Staubli VAL3: newProject1.dtx

public frame fUserFrame = {x=480, y=190, z=-101.4, rx=2, rz=-90, fatherId=world[0]}
public jointRx jtPark = {j1=-90, j2=-20, j3=130, j5=-60, j6=178}
public mdesc mNomSpeed = {blend=off}
public mdesc mdJointBlend = {accel=250, decel=150, leave=1, reach=1}
public mdesc mdLineBlend = {accel=80, vel=50, decel=50, tmax=100, rmax=9999, leave=2, reach=2}
public pointRx ptRoutingPath[478]
  [0] = {x=50.46, y=-3.411, z=224.779, rx=180, ry=-42.407, rz=-159.872, shoulder=lefty, elbow=epositive, wrist=wpositive, fatherId=fUserFrame[0]}
  [1] = {x=4.278, y=-3.411, z=174.216, rx=180, ry=-42.407, rz=-159.872, shoulder=lefty, elbow=epositive, wrist=wpositive, fatherId=fUserFrame[0]}
  [2] = {x=4.278, y=-3.411, z=124.216, rx=180, ry=-42.407, rz=-159.872, shoulder=lefty, elbow=epositive, wrist=wpositive, fatherId=fUserFrame[0]}
  [3] = {x=3.791, y=1.027, z=124.278, rx=180, ry=-42.212, rz=-156.401, shoulder=lefty, elbow=epositive, wrist=wpositive, fatherId=fUserFrame[0]}
  [4] = {x=4.289, y=5.504, z=124.132, rx=180, ry=-42.386, rz=-152.9, shoulder=lefty, elbow=epositive, wrist=wpositive, fatherId=fUserFrame[0]}
  [5] = {x=5.782, y=9.947, z=123.764, rx=180, ry=-42.934, rz=-149.41, shoulder=lefty, elbow=epositive, wrist=wpositive, fatherId=fUserFrame[0]}
  [6] = {x=8.224, y=14.41, z=123.139, rx=180, ry=-43.84, rz=-145.883, shoulder=lefty, elbow=epositive, wrist=wpositive, fatherId=fUserFrame[0]}
  [7] = {x=11.501, y=18.894, z=122.2, rx=180, ry=-45.057, rz=-142.303, shoulder=lefty, elbow=epositive, wrist=wpositive, fatherId=fUserFrame[0]}
  [8] = {x=9.824, y=14.861, z=122.959, rx=180, ry=-44.571, rz=-145.522, shoulder=lefty, elbow=epositive, wrist=wpositive, fatherId=fUserFrame[0]}
  [9] = {x=8.613, y=10.87, z=123.51, rx=180, ry=-44.23, rz=-148.678, shoulder=lefty, elbow=epositive, wrist=wpositive, fatherId=fUserFrame[0]}
  [10] = {x=7.921, y=6.919, z=123.87, rx=180, ry=-44.06, rz=-151.783, shoulder=lefty, elbow=epositive, wrist=wpositive, fatherId=fUserFrame[0]}
  [11] = {x=7.772, y=2.954, z=124.054, rx=180, ry=-44.073, rz=-154.884, shoulder=lefty, elbow=epositive, wrist=wpositive, fatherId=fUserFrame[0]}
  [12] = {x=8.16, y=-0.997, z=124.064, rx=180, ry=-44.266, rz=-157.97, shoulder=lefty, elbow=epositive, wrist=wpositive, fatherId=fUserFrame[0]}
  [13] = {x=7.987, y=2.551, z=124.05, rx=180, ry=-44.179, rz=-155.198, shoulder=lefty, elbow=epositive, wrist=wpositive, fatherId=fUserFrame[0]}
  [14] = {x=8.556, y=6.099, z=123.875, rx=180, ry=-44.383, rz=-152.423, shoulder=lefty, elbow=epositive, wrist=wpositive, fatherId=fUserFrame[0]}
  [15] = {x=9.86, y=9.613, z=123.529, rx=180, ry=-44.879, rz=-149.664, shoulder=lefty, elbow=epositive, wrist=wpositive, fatherId=fUserFrame[0]}
  [16] = {x=11.866, y=13.123, z=122.992, rx=180, ry=-45.653, rz=-146.893, shoulder=lefty, elbow=epositive, wrist=wpositive, fatherId=fUserFrame[0]}
  [17] = {x=14.502, y=16.628, z=122.234, rx=180, ry=-46.679, rz=-144.107, shoulder=lefty, elbow=epositive, wrist=wpositive, fatherId=fUserFrame[0]}
  [18] = {x=17.496, y=20.822, z=121.12, rx=180, ry=-47.769, rz=-140.737, shoulder=lefty, elbow=epositive, wrist=wpositive, fatherId=fUserFrame[0]}
  [19] = {x=20.739, y=24.824, z=119.755, rx=180, ry=-48.936, rz=-137.46, shoulder=lefty, elbow=epositive, wrist=wpositive, fatherId=fUserFrame[0]}
  [20] = {x=24.162, y=28.607, z=118.15, rx=180, ry=-50.165, rz=-134.293, shoulder=lefty, elbow=epositive, wrist=wpositive, fatherId=fUserFrame[0]}
  [21] = {x=27.716, y=32.196, z=116.305, rx=180, ry=-51.442, rz=-131.213, shoulder=lefty, elbow=epositive, wrist=wpositive, fatherId=fUserFrame[0]}
  [22] = {x=31.353, y=35.61, z=114.221, rx=180, ry=-52.756, rz=-128.203, shoulder=lefty, elbow=epositive, wrist=wpositive, fatherId=fUserFrame[0]}
  [23] = {x=35.033, y=38.861, z=111.903, rx=180, ry=-54.096, rz=-125.249, shoulder=lefty, elbow=epositive, wrist=wpositive, fatherId=fUserFrame[0]}
  [24] = {x=38.719, y=41.93, z=109.366, rx=180, ry=-55.456, rz=-122.365, shoulder=lefty, elbow=epositive, wrist=wpositive, fatherId=fUserFrame[0]}
  [25] = {x=42.278, y=44.785, z=106.677, rx=180, ry=-56.784, rz=-119.579, shoulder=lefty, elbow=epositive, wrist=wpositive, fatherId=fUserFrame[0]}
  [26] = {x=45.697, y=47.475, z=103.838, rx=180, ry=-58.069, rz=-116.85, shoulder=lefty, elbow=epositive, wrist=wpositive, fatherId=fUserFrame[0]}
  [27] = {x=49.013, y=50.027, z=100.834, rx=180, ry=-59.331, rz=-114.154, shoulder=lefty, elbow=epositive, wrist=wpositive, fatherId=fUserFrame[0]}
  [28] = {x=44.083, y=48.91, z=103.812, rx=180, ry=-56.777, rz=-115.386, shoulder=lefty, elbow=epositive, wrist=wpositive, fatherId=fUserFrame[0]}
  [29] = {x=38.578, y=47.741, z=106.69, rx=180, ry=-54.005, rz=-116.65, shoulder=lefty, elbow=epositive, wrist=wpositive, fatherId=fUserFrame[0]}
  [30] = {x=33.15, y=46.43, z=109.226, rx=180, ry=-51.395, rz=-118.029, shoulder=lefty, elbow=epositive, wrist=wpositive, fatherId=fUserFrame[0]}
  [31] = {x=27.673, y=45.016, z=111.467, rx=180, ry=-48.846, rz=-119.479, shoulder=lefty, elbow=epositive, wrist=wpositive, fatherId=fUserFrame[0]}
  [32] = {x=22.349, y=43.394, z=113.421, rx=180, ry=-46.48, rz=-121.092, shoulder=lefty, elbow=epositive, wrist=wpositive, fatherId=fUserFrame[0]}
  [33] = {x=16.731, y=41.59, z=115.171, rx=180, ry=-44.042, rz=-122.836, shoulder=lefty, elbow=epositive, wrist=wpositive, fatherId=fUserFrame[0]}
  [34] = {x=10.985, y=39.551, z=116.679, rx=180, ry=-41.623, rz=-124.751, shoulder=lefty, elbow=epositive, wrist=wpositive, fatherId=fUserFrame[0]}
  [35] = {x=5.01, y=37.376, z=117.894, rx=180, ry=-39.136, rz=-126.747, shoulder=lefty, elbow=epositive, wrist=wpositive, fatherId=fUserFrame[0]}
  [36] = {x=-0.804, y=35.019, z=118.802, rx=180, ry=-36.769, rz=-128.86, shoulder=lefty, elbow=epositive, wrist=wpositive, fatherId=fUserFrame[0]}
  [37] = {x=-6.341, y=32.513, z=119.42, rx=180, ry=-34.555, rz=-131.058, shoulder=lefty, elbow=epositive, wrist=wpositive, fatherId=fUserFrame[0]}
  [38] = {x=-11.541, y=29.826, z=119.795, rx=180, ry=-32.512, rz=-133.367, shoulder=lefty, elbow=epositive, wrist=wpositive, fatherId=fUserFrame[0]}
  [39] = {x=-16.328, y=26.961, z=119.972, rx=180, ry=-30.663, rz=-135.78, shoulder=lefty, elbow=epositive, wrist=wpositive, fatherId=fUserFrame[0]}
  [40] = {x=-20.759, y=23.89, z=119.984, rx=180, ry=-28.97, rz=-138.319, shoulder=lefty, elbow=epositive, wrist=wpositive, fatherId=fUserFrame[0]}
  [41] = {x=-24.662, y=20.615, z=119.891, rx=180, ry=-27.501, rz=-140.98, shoulder=lefty, elbow=epositive, wrist=wpositive, fatherId=fUserFrame[0]}
  [42] = {x=-28.137, y=17.281, z=119.682, rx=180, ry=-26.181, rz=-143.656, shoulder=lefty, elbow=epositive, wrist=wpositive, fatherId=fUserFrame[0]}
  [43] = {x=-30.954, y=14.026, z=119.435, rx=180, ry=-25.107, rz=-146.251, shoulder=lefty, elbow=epositive, wrist=wpositive, fatherId=fUserFrame[0]}
  [44] = {x=-33.378, y=10.884, z=119.125, rx=180, ry=-24.152, rz=-148.747, shoulder=lefty, elbow=epositive, wrist=wpositive, fatherId=fUserFrame[0]}
  [45] = {x=-35.18, y=7.837, z=118.856, rx=180, ry=-23.436, rz=-151.164, shoulder=lefty, elbow=epositive, wrist=wpositive, fatherId=fUserFrame[0]}
  [46] = {x=-36.701, y=4.771, z=118.561, rx=180, ry=-22.799, rz=-153.585, shoulder=lefty, elbow=epositive, wrist=wpositive, fatherId=fUserFrame[0]}
  [47] = {x=-37.634, y=1.68, z=118.351, rx=180, ry=-22.393, rz=-156.021, shoulder=lefty, elbow=epositive, wrist=wpositive, fatherId=fUserFrame[0]}
  [48] = {x=-31.685, y=1.329, z=120.133, rx=180, ry=-25.334, rz=-156.276, shoulder=lefty, elbow=epositive, wrist=wpositive, fatherId=fUserFrame[0]}
  [49] = {x=-28.486, y=1.091, z=120.955, rx=180, ry=-26.896, rz=-156.452, shoulder=lefty, elbow=epositive, wrist=wpositive, fatherId=fUserFrame[0]}
  [50] = {x=-25.13, y=0.851, z=121.716, rx=180, ry=-28.521, rz=-156.629, shoulder=lefty, elbow=epositive, wrist=wpositive, fatherId=fUserFrame[0]}
  [51] = {x=-21.648, y=0.56, z=122.401, rx=180, ry=-30.194, rz=-156.845, shoulder=lefty, elbow=epositive, wrist=wpositive, fatherId=fUserFrame[0]}
  [52] = {x=-17.999, y=0.268, z=123.005, rx=180, ry=-31.937, rz=-157.062, shoulder=lefty, elbow=epositive, wrist=wpositive, fatherId=fUserFrame[0]}
  [53] = {x=-14.2, y=-0.07, z=123.512, rx=180, ry=-33.74, rz=-157.314, shoulder=lefty, elbow=epositive, wrist=wpositive, fatherId=fUserFrame[0]}
  [54] = {x=-10.214, y=-0.41, z=123.912, rx=180, ry=-35.624, rz=-157.568, shoulder=lefty, elbow=epositive, wrist=wpositive, fatherId=fUserFrame[0]}
  [55] = {x=-6.064, y=-0.79, z=124.188, rx=180, ry=-37.576, rz=-157.852, shoulder=lefty, elbow=epositive, wrist=wpositive, fatherId=fUserFrame[0]}
  [56] = {x=-1.901, y=-1.162, z=124.321, rx=180, ry=-39.531, rz=-158.13, shoulder=lefty, elbow=epositive, wrist=wpositive, fatherId=fUserFrame[0]}
  [57] = {x=2.184, y=-1.553, z=124.312, rx=180, ry=-41.448, rz=-158.423, shoulder=lefty, elbow=epositive, wrist=wpositive, fatherId=fUserFrame[0]}
  [58] = {x=6.214, y=-1.935, z=124.167, rx=180, ry=-43.341, rz=-158.71, shoulder=lefty, elbow=epositive, wrist=wpositive, fatherId=fUserFrame[0]}
  [59] = {x=10.181, y=-2.334, z=123.892, rx=180, ry=-45.206, rz=-159.01, shoulder=lefty, elbow=epositive, wrist=wpositive, fatherId=fUserFrame[0]}
  [60] = {x=14.101, y=-2.726, z=123.491, rx=180, ry=-47.055, rz=-159.305, shoulder=lefty, elbow=epositive, wrist=wpositive, fatherId=fUserFrame[0]}
  [61] = {x=17.978, y=-3.133, z=122.966, rx=180, ry=-48.89, rz=-159.612, shoulder=lefty, elbow=epositive, wrist=wpositive, fatherId=fUserFrame[0]}
  [62] = {x=21.827, y=-3.535, z=122.317, rx=180, ry=-50.72, rz=-159.914, shoulder=lefty, elbow=epositive, wrist=wpositive, fatherId=fUserFrame[0]}
  [63] = {x=25.648, y=-3.944, z=121.544, rx=180, ry=-52.547, rz=-160.223, shoulder=lefty, elbow=epositive, wrist=wpositive, fatherId=fUserFrame[0]}
  [64] = {x=29.434, y=-4.346, z=120.65, rx=180, ry=-54.37, rz=-160.526, shoulder=lefty, elbow=epositive, wrist=wpositive, fatherId=fUserFrame[0]}
  [65] = {x=33.191, y=-4.75, z=119.634, rx=180, ry=-56.193, rz=-160.831, shoulder=lefty, elbow=epositive, wrist=wpositive, fatherId=fUserFrame[0]}
  [66] = {x=36.907, y=-5.147, z=118.499, rx=180, ry=-58.013, rz=-161.131, shoulder=lefty, elbow=epositive, wrist=wpositive, fatherId=fUserFrame[0]}
  [67] = {x=36.9, y=-1.421, z=118.608, rx=180, ry=-58.063, rz=-158.213, shoulder=lefty, elbow=epositive, wrist=wpositive, fatherId=fUserFrame[0]}
  [68] = {x=36.824, y=2.407, z=118.608, rx=180, ry=-58.029, rz=-155.227, shoulder=lefty, elbow=epositive, wrist=wpositive, fatherId=fUserFrame[0]}
  [69] = {x=36.718, y=6.276, z=118.48, rx=180, ry=-57.927, rz=-152.208, shoulder=lefty, elbow=epositive, wrist=wpositive, fatherId=fUserFrame[0]}
  [70] = {x=36.616, y=10.149, z=118.211, rx=180, ry=-57.771, rz=-149.173, shoulder=lefty, elbow=epositive, wrist=wpositive, fatherId=fUserFrame[0]}
  [71] = {x=36.51, y=14.016, z=117.804, rx=180, ry=-57.557, rz=-146.122, shoulder=lefty, elbow=epositive, wrist=wpositive, fatherId=fUserFrame[0]}
  [72] = {x=37.169, y=16.535, z=117.228, rx=180, ry=-57.751, rz=-144.116, shoulder=lefty, elbow=epositive, wrist=wpositive, fatherId=fUserFrame[0]}
  [73] = {x=38.02, y=19.029, z=116.525, rx=180, ry=-58.02, rz=-142.115, shoulder=lefty, elbow=epositive, wrist=wpositive, fatherId=fUserFrame[0]}
  [74] = {x=38.787, y=21.476, z=115.79, rx=180, ry=-58.228, rz=-140.133, shoulder=lefty, elbow=epositive, wrist=wpositive, fatherId=fUserFrame[0]}
  [75] = {x=39.708, y=23.854, z=114.947, rx=180, ry=-58.501, rz=-138.184, shoulder=lefty, elbow=epositive, wrist=wpositive, fatherId=fUserFrame[0]}
  [76] = {x=40.535, y=26.179, z=114.082, rx=180, ry=-58.709, rz=-136.254, shoulder=lefty, elbow=epositive, wrist=wpositive, fatherId=fUserFrame[0]}
  [77] = {x=41.497, y=28.44, z=113.115, rx=180, ry=-58.976, rz=-134.351, shoulder=lefty, elbow=epositive, wrist=wpositive, fatherId=fUserFrame[0]}
  [78] = {x=42.362, y=30.659, z=112.13, rx=180, ry=-59.176, rz=-132.457, shoulder=lefty, elbow=epositive, wrist=wpositive, fatherId=fUserFrame[0]}
  [79] = {x=43.343, y=32.818, z=111.05, rx=180, ry=-59.428, rz=-130.584, shoulder=lefty, elbow=epositive, wrist=wpositive, fatherId=fUserFrame[0]}
  [80] = {x=44.221, y=34.939, z=109.958, rx=180, ry=-59.61, rz=-128.715, shoulder=lefty, elbow=epositive, wrist=wpositive, fatherId=fUserFrame[0]}
  [81] = {x=45.196, y=37.004, z=108.778, rx=180, ry=-59.834, rz=-126.861, shoulder=lefty, elbow=epositive, wrist=wpositive, fatherId=fUserFrame[0]}
  [82] = {x=46.064, y=39.037, z=107.59, rx=180, ry=-59.985, rz=-125.002, shoulder=lefty, elbow=epositive, wrist=wpositive, fatherId=fUserFrame[0]}
  [83] = {x=47.013, y=41.002, z=106.326, rx=180, ry=-60.173, rz=-123.166, shoulder=lefty, elbow=epositive, wrist=wpositive, fatherId=fUserFrame[0]}
  [84] = {x=47.863, y=42.921, z=105.062, rx=180, ry=-60.293, rz=-121.334, shoulder=lefty, elbow=epositive, wrist=wpositive, fatherId=fUserFrame[0]}
  [85] = {x=48.809, y=44.772, z=103.716, rx=180, ry=-60.46, rz=-119.524, shoulder=lefty, elbow=epositive, wrist=wpositive, fatherId=fUserFrame[0]}
  [86] = {x=49.686, y=46.591, z=102.355, rx=180, ry=-60.572, rz=-117.702, shoulder=lefty, elbow=epositive, wrist=wpositive, fatherId=fUserFrame[0]}
  [87] = {x=50.7, y=48.352, z=100.888, rx=180, ry=-60.754, rz=-115.891, shoulder=lefty, elbow=epositive, wrist=wpositive, fatherId=fUserFrame[0]}
  [88] = {x=51.727, y=50.068, z=99.369, rx=180, ry=-60.931, rz=-114.077, shoulder=lefty, elbow=epositive, wrist=wpositive, fatherId=fUserFrame[0]}
  [89] = {x=52.948, y=51.706, z=97.716, rx=180, ry=-61.221, rz=-112.29, shoulder=lefty, elbow=epositive, wrist=wpositive, fatherId=fUserFrame[0]}
  [90] = {x=54.179, y=53.292, z=96.009, rx=180, ry=-61.51, rz=-110.505, shoulder=lefty, elbow=epositive, wrist=wpositive, fatherId=fUserFrame[0]}
  [91] = {x=55.616, y=54.796, z=94.148, rx=180, ry=-61.931, rz=-108.75, shoulder=lefty, elbow=epositive, wrist=wpositive, fatherId=fUserFrame[0]}
  [92] = {x=52.563, y=54.509, z=96.159, rx=180, ry=-60.128, rz=-109.12, shoulder=lefty, elbow=epositive, wrist=wpositive, fatherId=fUserFrame[0]}
  [93] = {x=47.423, y=53.901, z=99.331, rx=180, ry=-57.206, rz=-109.889, shoulder=lefty, elbow=epositive, wrist=wpositive, fatherId=fUserFrame[0]}
  [94] = {x=44.683, y=53.582, z=100.858, rx=180, ry=-55.691, rz=-110.285, shoulder=lefty, elbow=epositive, wrist=wpositive, fatherId=fUserFrame[0]}
  [95] = {x=41.917, y=53.209, z=102.324, rx=180, ry=-54.209, rz=-110.738, shoulder=lefty, elbow=epositive, wrist=wpositive, fatherId=fUserFrame[0]}
  [96] = {x=38.974, y=52.828, z=103.762, rx=180, ry=-52.655, rz=-111.197, shoulder=lefty, elbow=epositive, wrist=wpositive, fatherId=fUserFrame[0]}
  [97] = {x=36.005, y=52.436, z=105.108, rx=180, ry=-51.115, rz=-111.665, shoulder=lefty, elbow=epositive, wrist=wpositive, fatherId=fUserFrame[0]}
  [98] = {x=33.04, y=52.03, z=106.355, rx=180, ry=-49.603, rz=-112.143, shoulder=lefty, elbow=epositive, wrist=wpositive, fatherId=fUserFrame[0]}
  [99] = {x=27.328, y=51.09, z=108.557, rx=180, ry=-46.799, rz=-113.223, shoulder=lefty, elbow=epositive, wrist=wpositive, fatherId=fUserFrame[0]}
  [100] = {x=21.384, y=50.082, z=110.477, rx=180, ry=-43.956, rz=-114.355, shoulder=lefty, elbow=epositive, wrist=wpositive, fatherId=fUserFrame[0]}
  [101] = {x=18.339, y=49.516, z=111.339, rx=180, ry=-42.539, rz=-114.977, shoulder=lefty, elbow=epositive, wrist=wpositive, fatherId=fUserFrame[0]}
  [102] = {x=15.169, y=48.922, z=112.135, rx=180, ry=-41.078, rz=-115.621, shoulder=lefty, elbow=epositive, wrist=wpositive, fatherId=fUserFrame[0]}
  [103] = {x=11.868, y=48.297, z=112.858, rx=180, ry=-39.57, rz=-116.289, shoulder=lefty, elbow=epositive, wrist=wpositive, fatherId=fUserFrame[0]}
  [104] = {x=8.507, y=47.631, z=113.495, rx=180, ry=-38.055, rz=-116.989, shoulder=lefty, elbow=epositive, wrist=wpositive, fatherId=fUserFrame[0]}
  [105] = {x=5.171, y=46.89, z=114.053, rx=180, ry=-36.584, rz=-117.755, shoulder=lefty, elbow=epositive, wrist=wpositive, fatherId=fUserFrame[0]}
  [106] = {x=1.817, y=46.093, z=114.527, rx=180, ry=-35.126, rz=-118.565, shoulder=lefty, elbow=epositive, wrist=wpositive, fatherId=fUserFrame[0]}
  [107] = {x=-1.542, y=45.234, z=114.917, rx=180, ry=-33.688, rz=-119.423, shoulder=lefty, elbow=epositive, wrist=wpositive, fatherId=fUserFrame[0]}
  [108] = {x=-4.897, y=44.308, z=115.225, rx=180, ry=-32.273, rz=-120.333, shoulder=lefty, elbow=epositive, wrist=wpositive, fatherId=fUserFrame[0]}
  [109] = {x=-11.566, y=42.2, z=115.614, rx=180, ry=-29.532, rz=-122.352, shoulder=lefty, elbow=epositive, wrist=wpositive, fatherId=fUserFrame[0]}
  [110] = {x=-17.965, y=39.906, z=115.675, rx=180, ry=-26.955, rz=-124.491, shoulder=lefty, elbow=epositive, wrist=wpositive, fatherId=fUserFrame[0]}
  [111] = {x=-24.031, y=37.42, z=115.459, rx=180, ry=-24.556, rz=-126.753, shoulder=lefty, elbow=epositive, wrist=wpositive, fatherId=fUserFrame[0]}
  [112] = {x=-29.593, y=34.771, z=115.041, rx=180, ry=-22.399, rz=-129.107, shoulder=lefty, elbow=epositive, wrist=wpositive, fatherId=fUserFrame[0]}
  [113] = {x=-34.725, y=31.939, z=114.463, rx=180, ry=-20.436, rz=-131.569, shoulder=lefty, elbow=epositive, wrist=wpositive, fatherId=fUserFrame[0]}
  [114] = {x=-39.297, y=28.891, z=113.822, rx=180, ry=-18.731, rz=-134.16, shoulder=lefty, elbow=epositive, wrist=wpositive, fatherId=fUserFrame[0]}
  [115] = {x=-43.448, y=25.6, z=113.12, rx=180, ry=-17.202, rz=-136.9, shoulder=lefty, elbow=epositive, wrist=wpositive, fatherId=fUserFrame[0]}
  [116] = {x=-47.036, y=22.037, z=112.449, rx=180, ry=-15.915, rz=-139.808, shoulder=lefty, elbow=epositive, wrist=wpositive, fatherId=fUserFrame[0]}
  [117] = {x=-50.183, y=18.336, z=111.758, rx=180, ry=-14.774, rz=-142.782, shoulder=lefty, elbow=epositive, wrist=wpositive, fatherId=fUserFrame[0]}
  [118] = {x=-52.715, y=14.806, z=111.116, rx=180, ry=-13.835, rz=-145.601, shoulder=lefty, elbow=epositive, wrist=wpositive, fatherId=fUserFrame[0]}
  [119] = {x=-52.715, y=14.806, z=161.116, rx=180, ry=-13.835, rz=-145.601, shoulder=lefty, elbow=epositive, wrist=wpositive, fatherId=fUserFrame[0]}
  [120] = {x=4.278, y=3.411, z=174.216, rx=180, ry=-42.407, rz=159.872, shoulder=lefty, elbow=epositive, wrist=wpositive, fatherId=fUserFrame[0]}
  [121] = {x=4.278, y=3.411, z=124.216, rx=180, ry=-42.407, rz=159.872, shoulder=lefty, elbow=epositive, wrist=wpositive, fatherId=fUserFrame[0]}
  [122] = {x=3.791, y=-1.027, z=124.278, rx=180, ry=-42.212, rz=156.401, shoulder=lefty, elbow=epositive, wrist=wpositive, fatherId=fUserFrame[0]}
  [123] = {x=4.289, y=-5.504, z=124.132, rx=180, ry=-42.386, rz=152.9, shoulder=lefty, elbow=epositive, wrist=wpositive, fatherId=fUserFrame[0]}
  [124] = {x=5.782, y=-9.947, z=123.764, rx=180, ry=-42.934, rz=149.41, shoulder=lefty, elbow=epositive, wrist=wpositive, fatherId=fUserFrame[0]}
  [125] = {x=8.224, y=-14.41, z=123.139, rx=180, ry=-43.84, rz=145.883, shoulder=lefty, elbow=epositive, wrist=wpositive, fatherId=fUserFrame[0]}
  [126] = {x=11.501, y=-18.894, z=122.2, rx=180, ry=-45.057, rz=142.303, shoulder=lefty, elbow=epositive, wrist=wpositive, fatherId=fUserFrame[0]}
  [127] = {x=9.824, y=-14.861, z=122.959, rx=180, ry=-44.571, rz=145.522, shoulder=lefty, elbow=epositive, wrist=wpositive, fatherId=fUserFrame[0]}
  [128] = {x=8.613, y=-10.87, z=123.51, rx=180, ry=-44.23, rz=148.678, shoulder=lefty, elbow=epositive, wrist=wpositive, fatherId=fUserFrame[0]}
  [129] = {x=7.921, y=-6.919, z=123.87, rx=180, ry=-44.06, rz=151.783, shoulder=lefty, elbow=epositive, wrist=wpositive, fatherId=fUserFrame[0]}
  [130] = {x=7.772, y=-2.954, z=124.054, rx=180, ry=-44.073, rz=154.884, shoulder=lefty, elbow=epositive, wrist=wpositive, fatherId=fUserFrame[0]}
  [131] = {x=8.16, y=0.997, z=124.064, rx=180, ry=-44.266, rz=157.97, shoulder=lefty, elbow=epositive, wrist=wpositive, fatherId=fUserFrame[0]}
  [132] = {x=7.987, y=-2.551, z=124.05, rx=180, ry=-44.179, rz=155.198, shoulder=lefty, elbow=epositive, wrist=wpositive, fatherId=fUserFrame[0]}
  [133] = {x=8.556, y=-6.099, z=123.875, rx=180, ry=-44.383, rz=152.423, shoulder=lefty, elbow=epositive, wrist=wpositive, fatherId=fUserFrame[0]}
  [134] = {x=9.86, y=-9.613, z=123.529, rx=180, ry=-44.879, rz=149.664, shoulder=lefty, elbow=epositive, wrist=wpositive, fatherId=fUserFrame[0]}
  [135] = {x=11.866, y=-13.123, z=122.992, rx=180, ry=-45.653, rz=146.893, shoulder=lefty, elbow=epositive, wrist=wpositive, fatherId=fUserFrame[0]}
  [136] = {x=14.502, y=-16.628, z=122.234, rx=180, ry=-46.679, rz=144.107, shoulder=lefty, elbow=epositive, wrist=wpositive, fatherId=fUserFrame[0]}
  [137] = {x=17.496, y=-20.822, z=121.12, rx=180, ry=-47.769, rz=140.737, shoulder=lefty, elbow=epositive, wrist=wpositive, fatherId=fUserFrame[0]}
  [138] = {x=20.739, y=-24.824, z=119.755, rx=180, ry=-48.936, rz=137.46, shoulder=lefty, elbow=epositive, wrist=wpositive, fatherId=fUserFrame[0]}
  [139] = {x=24.162, y=-28.607, z=118.15, rx=180, ry=-50.165, rz=134.293, shoulder=lefty, elbow=epositive, wrist=wpositive, fatherId=fUserFrame[0]}
  [140] = {x=27.716, y=-32.196, z=116.305, rx=180, ry=-51.442, rz=131.213, shoulder=lefty, elbow=epositive, wrist=wpositive, fatherId=fUserFrame[0]}
  [141] = {x=31.353, y=-35.61, z=114.221, rx=180, ry=-52.756, rz=128.203, shoulder=lefty, elbow=epositive, wrist=wpositive, fatherId=fUserFrame[0]}
  [142] = {x=35.033, y=-38.861, z=111.903, rx=180, ry=-54.096, rz=125.249, shoulder=lefty, elbow=epositive, wrist=wpositive, fatherId=fUserFrame[0]}
  [143] = {x=38.719, y=-41.93, z=109.366, rx=180, ry=-55.456, rz=122.365, shoulder=lefty, elbow=epositive, wrist=wpositive, fatherId=fUserFrame[0]}
  [144] = {x=42.278, y=-44.785, z=106.677, rx=180, ry=-56.784, rz=119.579, shoulder=lefty, elbow=epositive, wrist=wpositive, fatherId=fUserFrame[0]}
  [145] = {x=45.697, y=-47.475, z=103.838, rx=180, ry=-58.069, rz=116.85, shoulder=lefty, elbow=epositive, wrist=wpositive, fatherId=fUserFrame[0]}
  [146] = {x=49.013, y=-50.027, z=100.834, rx=180, ry=-59.331, rz=114.154, shoulder=lefty, elbow=epositive, wrist=wpositive, fatherId=fUserFrame[0]}
  [147] = {x=44.083, y=-48.91, z=103.812, rx=180, ry=-56.777, rz=115.386, shoulder=lefty, elbow=epositive, wrist=wpositive, fatherId=fUserFrame[0]}
  [148] = {x=38.578, y=-47.741, z=106.69, rx=180, ry=-54.005, rz=116.65, shoulder=lefty, elbow=epositive, wrist=wpositive, fatherId=fUserFrame[0]}
  [149] = {x=33.15, y=-46.43, z=109.226, rx=180, ry=-51.395, rz=118.029, shoulder=lefty, elbow=epositive, wrist=wpositive, fatherId=fUserFrame[0]}
  [150] = {x=27.673, y=-45.016, z=111.467, rx=180, ry=-48.846, rz=119.479, shoulder=lefty, elbow=epositive, wrist=wpositive, fatherId=fUserFrame[0]}
  [151] = {x=22.349, y=-43.394, z=113.421, rx=180, ry=-46.48, rz=121.092, shoulder=lefty, elbow=epositive, wrist=wpositive, fatherId=fUserFrame[0]}
  [152] = {x=16.731, y=-41.59, z=115.171, rx=180, ry=-44.042, rz=122.836, shoulder=lefty, elbow=epositive, wrist=wpositive, fatherId=fUserFrame[0]}
  [153] = {x=10.985, y=-39.551, z=116.679, rx=180, ry=-41.623, rz=124.751, shoulder=lefty, elbow=epositive, wrist=wpositive, fatherId=fUserFrame[0]}
  [154] = {x=5.01, y=-37.376, z=117.894, rx=180, ry=-39.136, rz=126.747, shoulder=lefty, elbow=epositive, wrist=wpositive, fatherId=fUserFrame[0]}
  [155] = {x=-0.804, y=-35.019, z=118.802, rx=180, ry=-36.769, rz=128.86, shoulder=lefty, elbow=epositive, wrist=wpositive, fatherId=fUserFrame[0]}
  [156] = {x=-6.341, y=-32.513, z=119.42, rx=180, ry=-34.555, rz=131.058, shoulder=lefty, elbow=epositive, wrist=wpositive, fatherId=fUserFrame[0]}
  [157] = {x=-11.541, y=-29.826, z=119.795, rx=180, ry=-32.512, rz=133.367, shoulder=lefty, elbow=epositive, wrist=wpositive, fatherId=fUserFrame[0]}
  [158] = {x=-16.328, y=-26.961, z=119.972, rx=180, ry=-30.663, rz=135.78, shoulder=lefty, elbow=epositive, wrist=wpositive, fatherId=fUserFrame[0]}
  [159] = {x=-20.759, y=-23.89, z=119.984, rx=180, ry=-28.97, rz=138.319, shoulder=lefty, elbow=epositive, wrist=wpositive, fatherId=fUserFrame[0]}
  [160] = {x=-24.662, y=-20.615, z=119.891, rx=180, ry=-27.501, rz=140.98, shoulder=lefty, elbow=epositive, wrist=wpositive, fatherId=fUserFrame[0]}
  [161] = {x=-28.137, y=-17.281, z=119.682, rx=180, ry=-26.181, rz=143.656, shoulder=lefty, elbow=epositive, wrist=wpositive, fatherId=fUserFrame[0]}
  [162] = {x=-30.954, y=-14.026, z=119.435, rx=180, ry=-25.107, rz=146.251, shoulder=lefty, elbow=epositive, wrist=wpositive, fatherId=fUserFrame[0]}
  [163] = {x=-33.378, y=-10.884, z=119.125, rx=180, ry=-24.152, rz=148.747, shoulder=lefty, elbow=epositive, wrist=wpositive, fatherId=fUserFrame[0]}
  [164] = {x=-35.18, y=-7.837, z=118.856, rx=180, ry=-23.436, rz=151.164, shoulder=lefty, elbow=epositive, wrist=wpositive, fatherId=fUserFrame[0]}
  [165] = {x=-36.701, y=-4.771, z=118.561, rx=180, ry=-22.799, rz=153.585, shoulder=lefty, elbow=epositive, wrist=wpositive, fatherId=fUserFrame[0]}
  [166] = {x=-37.634, y=-1.68, z=118.351, rx=180, ry=-22.393, rz=156.021, shoulder=lefty, elbow=epositive, wrist=wpositive, fatherId=fUserFrame[0]}
  [167] = {x=-31.685, y=-1.329, z=120.133, rx=180, ry=-25.334, rz=156.276, shoulder=lefty, elbow=epositive, wrist=wpositive, fatherId=fUserFrame[0]}
  [168] = {x=-28.486, y=-1.091, z=120.955, rx=180, ry=-26.896, rz=156.452, shoulder=lefty, elbow=epositive, wrist=wpositive, fatherId=fUserFrame[0]}
  [169] = {x=-25.13, y=-0.851, z=121.716, rx=180, ry=-28.521, rz=156.629, shoulder=lefty, elbow=epositive, wrist=wpositive, fatherId=fUserFrame[0]}
  [170] = {x=-21.648, y=-0.56, z=122.401, rx=180, ry=-30.194, rz=156.845, shoulder=lefty, elbow=epositive, wrist=wpositive, fatherId=fUserFrame[0]}
  [171] = {x=-17.999, y=-0.268, z=123.005, rx=180, ry=-31.937, rz=157.062, shoulder=lefty, elbow=epositive, wrist=wpositive, fatherId=fUserFrame[0]}
  [172] = {x=-14.2, y=0.07, z=123.512, rx=180, ry=-33.74, rz=157.314, shoulder=lefty, elbow=epositive, wrist=wpositive, fatherId=fUserFrame[0]}
  [173] = {x=-10.214, y=0.41, z=123.912, rx=180, ry=-35.624, rz=157.568, shoulder=lefty, elbow=epositive, wrist=wpositive, fatherId=fUserFrame[0]}
  [174] = {x=-6.064, y=0.79, z=124.188, rx=180, ry=-37.576, rz=157.852, shoulder=lefty, elbow=epositive, wrist=wpositive, fatherId=fUserFrame[0]}
  [175] = {x=-1.901, y=1.162, z=124.321, rx=180, ry=-39.531, rz=158.13, shoulder=lefty, elbow=epositive, wrist=wpositive, fatherId=fUserFrame[0]}
  [176] = {x=2.184, y=1.553, z=124.312, rx=180, ry=-41.448, rz=158.423, shoulder=lefty, elbow=epositive, wrist=wpositive, fatherId=fUserFrame[0]}
  [177] = {x=6.214, y=1.935, z=124.167, rx=180, ry=-43.341, rz=158.71, shoulder=lefty, elbow=epositive, wrist=wpositive, fatherId=fUserFrame[0]}
  [178] = {x=10.181, y=2.334, z=123.892, rx=180, ry=-45.206, rz=159.01, shoulder=lefty, elbow=epositive, wrist=wpositive, fatherId=fUserFrame[0]}
  [179] = {x=14.101, y=2.726, z=123.491, rx=180, ry=-47.055, rz=159.305, shoulder=lefty, elbow=epositive, wrist=wpositive, fatherId=fUserFrame[0]}
  [180] = {x=17.978, y=3.133, z=122.966, rx=180, ry=-48.89, rz=159.612, shoulder=lefty, elbow=epositive, wrist=wpositive, fatherId=fUserFrame[0]}
  [181] = {x=21.827, y=3.535, z=122.317, rx=180, ry=-50.72, rz=159.914, shoulder=lefty, elbow=epositive, wrist=wpositive, fatherId=fUserFrame[0]}
  [182] = {x=25.648, y=3.944, z=121.544, rx=180, ry=-52.547, rz=160.223, shoulder=lefty, elbow=epositive, wrist=wpositive, fatherId=fUserFrame[0]}
  [183] = {x=29.434, y=4.346, z=120.65, rx=180, ry=-54.37, rz=160.526, shoulder=lefty, elbow=epositive, wrist=wpositive, fatherId=fUserFrame[0]}
  [184] = {x=33.191, y=4.75, z=119.634, rx=180, ry=-56.193, rz=160.831, shoulder=lefty, elbow=epositive, wrist=wpositive, fatherId=fUserFrame[0]}
  [185] = {x=36.907, y=5.147, z=118.499, rx=180, ry=-58.013, rz=161.131, shoulder=lefty, elbow=epositive, wrist=wpositive, fatherId=fUserFrame[0]}
  [186] = {x=36.9, y=1.421, z=118.608, rx=180, ry=-58.063, rz=158.213, shoulder=lefty, elbow=epositive, wrist=wpositive, fatherId=fUserFrame[0]}
  [187] = {x=36.824, y=-2.407, z=118.608, rx=180, ry=-58.029, rz=155.227, shoulder=lefty, elbow=epositive, wrist=wpositive, fatherId=fUserFrame[0]}
  [188] = {x=36.718, y=-6.276, z=118.48, rx=180, ry=-57.927, rz=152.208, shoulder=lefty, elbow=epositive, wrist=wpositive, fatherId=fUserFrame[0]}
  [189] = {x=36.616, y=-10.149, z=118.211, rx=180, ry=-57.771, rz=149.173, shoulder=lefty, elbow=epositive, wrist=wpositive, fatherId=fUserFrame[0]}
  [190] = {x=36.51, y=-14.016, z=117.804, rx=180, ry=-57.557, rz=146.122, shoulder=lefty, elbow=epositive, wrist=wpositive, fatherId=fUserFrame[0]}
  [191] = {x=37.169, y=-16.535, z=117.228, rx=180, ry=-57.751, rz=144.116, shoulder=lefty, elbow=epositive, wrist=wpositive, fatherId=fUserFrame[0]}
  [192] = {x=38.02, y=-19.029, z=116.525, rx=180, ry=-58.02, rz=142.115, shoulder=lefty, elbow=epositive, wrist=wpositive, fatherId=fUserFrame[0]}
  [193] = {x=38.787, y=-21.476, z=115.79, rx=180, ry=-58.228, rz=140.133, shoulder=lefty, elbow=epositive, wrist=wpositive, fatherId=fUserFrame[0]}
  [194] = {x=39.708, y=-23.854, z=114.947, rx=180, ry=-58.501, rz=138.184, shoulder=lefty, elbow=epositive, wrist=wpositive, fatherId=fUserFrame[0]}
  [195] = {x=40.535, y=-26.179, z=114.082, rx=180, ry=-58.709, rz=136.254, shoulder=lefty, elbow=epositive, wrist=wpositive, fatherId=fUserFrame[0]}
  [196] = {x=41.497, y=-28.44, z=113.115, rx=180, ry=-58.976, rz=134.351, shoulder=lefty, elbow=epositive, wrist=wpositive, fatherId=fUserFrame[0]}
  [197] = {x=42.362, y=-30.659, z=112.13, rx=180, ry=-59.176, rz=132.457, shoulder=lefty, elbow=epositive, wrist=wpositive, fatherId=fUserFrame[0]}
  [198] = {x=43.343, y=-32.818, z=111.05, rx=180, ry=-59.428, rz=130.584, shoulder=lefty, elbow=epositive, wrist=wpositive, fatherId=fUserFrame[0]}
  [199] = {x=44.221, y=-34.939, z=109.958, rx=180, ry=-59.61, rz=128.715, shoulder=lefty, elbow=epositive, wrist=wpositive, fatherId=fUserFrame[0]}
  [200] = {x=45.196, y=-37.004, z=108.778, rx=180, ry=-59.834, rz=126.861, shoulder=lefty, elbow=epositive, wrist=wpositive, fatherId=fUserFrame[0]}
  [201] = {x=46.064, y=-39.037, z=107.59, rx=180, ry=-59.985, rz=125.002, shoulder=lefty, elbow=epositive, wrist=wpositive, fatherId=fUserFrame[0]}
  [202] = {x=47.013, y=-41.002, z=106.326, rx=180, ry=-60.173, rz=123.166, shoulder=lefty, elbow=epositive, wrist=wpositive, fatherId=fUserFrame[0]}
  [203] = {x=47.863, y=-42.921, z=105.062, rx=180, ry=-60.293, rz=121.334, shoulder=lefty, elbow=epositive, wrist=wpositive, fatherId=fUserFrame[0]}
  [204] = {x=48.809, y=-44.772, z=103.716, rx=180, ry=-60.46, rz=119.524, shoulder=lefty, elbow=epositive, wrist=wpositive, fatherId=fUserFrame[0]}
  [205] = {x=49.686, y=-46.591, z=102.355, rx=180, ry=-60.572, rz=117.702, shoulder=lefty, elbow=epositive, wrist=wpositive, fatherId=fUserFrame[0]}
  [206] = {x=50.7, y=-48.352, z=100.888, rx=180, ry=-60.754, rz=115.891, shoulder=lefty, elbow=epositive, wrist=wpositive, fatherId=fUserFrame[0]}
  [207] = {x=51.727, y=-50.068, z=99.369, rx=180, ry=-60.931, rz=114.077, shoulder=lefty, elbow=epositive, wrist=wpositive, fatherId=fUserFrame[0]}
  [208] = {x=52.948, y=-51.706, z=97.716, rx=180, ry=-61.221, rz=112.29, shoulder=lefty, elbow=epositive, wrist=wpositive, fatherId=fUserFrame[0]}
  [209] = {x=54.179, y=-53.292, z=96.009, rx=180, ry=-61.51, rz=110.505, shoulder=lefty, elbow=epositive, wrist=wpositive, fatherId=fUserFrame[0]}
  [210] = {x=55.616, y=-54.796, z=94.148, rx=180, ry=-61.931, rz=108.75, shoulder=lefty, elbow=epositive, wrist=wpositive, fatherId=fUserFrame[0]}
  [211] = {x=52.563, y=-54.509, z=96.159, rx=180, ry=-60.128, rz=109.12, shoulder=lefty, elbow=epositive, wrist=wpositive, fatherId=fUserFrame[0]}
  [212] = {x=47.423, y=-53.901, z=99.331, rx=180, ry=-57.206, rz=109.889, shoulder=lefty, elbow=epositive, wrist=wpositive, fatherId=fUserFrame[0]}
  [213] = {x=44.683, y=-53.582, z=100.858, rx=180, ry=-55.691, rz=110.285, shoulder=lefty, elbow=epositive, wrist=wpositive, fatherId=fUserFrame[0]}
  [214] = {x=41.917, y=-53.209, z=102.324, rx=180, ry=-54.209, rz=110.738, shoulder=lefty, elbow=epositive, wrist=wpositive, fatherId=fUserFrame[0]}
  [215] = {x=38.974, y=-52.828, z=103.762, rx=180, ry=-52.655, rz=111.197, shoulder=lefty, elbow=epositive, wrist=wpositive, fatherId=fUserFrame[0]}
  [216] = {x=36.005, y=-52.436, z=105.108, rx=180, ry=-51.115, rz=111.665, shoulder=lefty, elbow=epositive, wrist=wpositive, fatherId=fUserFrame[0]}
  [217] = {x=33.04, y=-52.03, z=106.355, rx=180, ry=-49.603, rz=112.143, shoulder=lefty, elbow=epositive, wrist=wpositive, fatherId=fUserFrame[0]}
  [218] = {x=27.328, y=-51.09, z=108.557, rx=180, ry=-46.799, rz=113.223, shoulder=lefty, elbow=epositive, wrist=wpositive, fatherId=fUserFrame[0]}
  [219] = {x=21.384, y=-50.082, z=110.477, rx=180, ry=-43.956, rz=114.355, shoulder=lefty, elbow=epositive, wrist=wpositive, fatherId=fUserFrame[0]}
  [220] = {x=18.339, y=-49.516, z=111.339, rx=180, ry=-42.539, rz=114.977, shoulder=lefty, elbow=epositive, wrist=wpositive, fatherId=fUserFrame[0]}
  [221] = {x=15.169, y=-48.922, z=112.135, rx=180, ry=-41.078, rz=115.621, shoulder=lefty, elbow=epositive, wrist=wpositive, fatherId=fUserFrame[0]}
  [222] = {x=11.868, y=-48.297, z=112.858, rx=180, ry=-39.57, rz=116.289, shoulder=lefty, elbow=epositive, wrist=wpositive, fatherId=fUserFrame[0]}
  [223] = {x=8.507, y=-47.631, z=113.495, rx=180, ry=-38.055, rz=116.989, shoulder=lefty, elbow=epositive, wrist=wpositive, fatherId=fUserFrame[0]}
  [224] = {x=5.171, y=-46.89, z=114.053, rx=180, ry=-36.584, rz=117.755, shoulder=lefty, elbow=epositive, wrist=wpositive, fatherId=fUserFrame[0]}
  [225] = {x=1.817, y=-46.093, z=114.527, rx=180, ry=-35.126, rz=118.565, shoulder=lefty, elbow=epositive, wrist=wpositive, fatherId=fUserFrame[0]}
  [226] = {x=-1.542, y=-45.234, z=114.917, rx=180, ry=-33.688, rz=119.423, shoulder=lefty, elbow=epositive, wrist=wpositive, fatherId=fUserFrame[0]}
  [227] = {x=-4.897, y=-44.308, z=115.225, rx=180, ry=-32.273, rz=120.333, shoulder=lefty, elbow=epositive, wrist=wpositive, fatherId=fUserFrame[0]}
  [228] = {x=-11.566, y=-42.2, z=115.614, rx=180, ry=-29.532, rz=122.352, shoulder=lefty, elbow=epositive, wrist=wpositive, fatherId=fUserFrame[0]}
  [229] = {x=-17.965, y=-39.906, z=115.675, rx=180, ry=-26.955, rz=124.491, shoulder=lefty, elbow=epositive, wrist=wpositive, fatherId=fUserFrame[0]}
  [230] = {x=-24.031, y=-37.42, z=115.459, rx=180, ry=-24.556, rz=126.753, shoulder=lefty, elbow=epositive, wrist=wpositive, fatherId=fUserFrame[0]}
  [231] = {x=-29.593, y=-34.771, z=115.041, rx=180, ry=-22.399, rz=129.107, shoulder=lefty, elbow=epositive, wrist=wpositive, fatherId=fUserFrame[0]}
  [232] = {x=-34.725, y=-31.939, z=114.463, rx=180, ry=-20.436, rz=131.569, shoulder=lefty, elbow=epositive, wrist=wpositive, fatherId=fUserFrame[0]}
  [233] = {x=-39.297, y=-28.891, z=113.822, rx=180, ry=-18.731, rz=134.16, shoulder=lefty, elbow=epositive, wrist=wpositive, fatherId=fUserFrame[0]}
  [234] = {x=-43.448, y=-25.6, z=113.12, rx=180, ry=-17.202, rz=136.9, shoulder=lefty, elbow=epositive, wrist=wpositive, fatherId=fUserFrame[0]}
  [235] = {x=-47.036, y=-22.037, z=112.449, rx=180, ry=-15.915, rz=139.808, shoulder=lefty, elbow=epositive, wrist=wpositive, fatherId=fUserFrame[0]}
  [236] = {x=-50.183, y=-18.336, z=111.758, rx=180, ry=-14.774, rz=142.782, shoulder=lefty, elbow=epositive, wrist=wpositive, fatherId=fUserFrame[0]}
  [237] = {x=-52.715, y=-14.806, z=111.116, rx=180, ry=-13.835, rz=145.601, shoulder=lefty, elbow=epositive, wrist=wpositive, fatherId=fUserFrame[0]}
  [238] = {x=-52.715, y=-14.806, z=161.116, rx=180, ry=-13.835, rz=145.601, shoulder=lefty, elbow=epositive, wrist=wpositive, fatherId=fUserFrame[0]}
  [239] = {x=4.278, y=-3.411, z=174.216, rx=180, ry=-42.407, rz=20.128, shoulder=lefty, elbow=epositive, wrist=wpositive, fatherId=fUserFrame[0]}
  [240] = {x=4.278, y=-3.411, z=124.216, rx=180, ry=-42.407, rz=20.128, shoulder=lefty, elbow=epositive, wrist=wpositive, fatherId=fUserFrame[0]}
  [241] = {x=3.791, y=1.027, z=124.278, rx=180, ry=-42.212, rz=23.599, shoulder=lefty, elbow=epositive, wrist=wpositive, fatherId=fUserFrame[0]}
  [242] = {x=4.289, y=5.504, z=124.132, rx=180, ry=-42.386, rz=27.1, shoulder=lefty, elbow=epositive, wrist=wpositive, fatherId=fUserFrame[0]}
  [243] = {x=5.782, y=9.947, z=123.764, rx=180, ry=-42.934, rz=30.59, shoulder=lefty, elbow=epositive, wrist=wpositive, fatherId=fUserFrame[0]}
  [244] = {x=8.224, y=14.41, z=123.139, rx=180, ry=-43.84, rz=34.117, shoulder=lefty, elbow=epositive, wrist=wpositive, fatherId=fUserFrame[0]}
  [245] = {x=11.501, y=18.894, z=122.2, rx=180, ry=-45.057, rz=37.697, shoulder=lefty, elbow=epositive, wrist=wpositive, fatherId=fUserFrame[0]}
  [246] = {x=9.824, y=14.861, z=122.959, rx=180, ry=-44.571, rz=34.478, shoulder=lefty, elbow=epositive, wrist=wpositive, fatherId=fUserFrame[0]}
  [247] = {x=8.613, y=10.87, z=123.51, rx=180, ry=-44.23, rz=31.322, shoulder=lefty, elbow=epositive, wrist=wpositive, fatherId=fUserFrame[0]}
  [248] = {x=7.921, y=6.919, z=123.87, rx=180, ry=-44.06, rz=28.217, shoulder=lefty, elbow=epositive, wrist=wpositive, fatherId=fUserFrame[0]}
  [249] = {x=7.772, y=2.954, z=124.054, rx=180, ry=-44.073, rz=25.116, shoulder=lefty, elbow=epositive, wrist=wpositive, fatherId=fUserFrame[0]}
  [250] = {x=8.16, y=-0.997, z=124.064, rx=180, ry=-44.266, rz=22.03, shoulder=lefty, elbow=epositive, wrist=wpositive, fatherId=fUserFrame[0]}
  [251] = {x=7.987, y=2.551, z=124.05, rx=180, ry=-44.179, rz=24.802, shoulder=lefty, elbow=epositive, wrist=wpositive, fatherId=fUserFrame[0]}
  [252] = {x=8.556, y=6.099, z=123.875, rx=180, ry=-44.383, rz=27.577, shoulder=lefty, elbow=epositive, wrist=wpositive, fatherId=fUserFrame[0]}
  [253] = {x=9.86, y=9.613, z=123.529, rx=180, ry=-44.879, rz=30.336, shoulder=lefty, elbow=epositive, wrist=wpositive, fatherId=fUserFrame[0]}
  [254] = {x=11.866, y=13.123, z=122.992, rx=180, ry=-45.653, rz=33.107, shoulder=lefty, elbow=epositive, wrist=wpositive, fatherId=fUserFrame[0]}
  [255] = {x=14.502, y=16.628, z=122.234, rx=180, ry=-46.679, rz=35.893, shoulder=lefty, elbow=epositive, wrist=wpositive, fatherId=fUserFrame[0]}
  [256] = {x=17.496, y=20.822, z=121.12, rx=180, ry=-47.769, rz=39.263, shoulder=lefty, elbow=epositive, wrist=wpositive, fatherId=fUserFrame[0]}
  [257] = {x=20.739, y=24.824, z=119.755, rx=180, ry=-48.936, rz=42.54, shoulder=lefty, elbow=epositive, wrist=wpositive, fatherId=fUserFrame[0]}
  [258] = {x=24.162, y=28.607, z=118.15, rx=180, ry=-50.165, rz=45.707, shoulder=lefty, elbow=epositive, wrist=wpositive, fatherId=fUserFrame[0]}
  [259] = {x=27.716, y=32.196, z=116.305, rx=180, ry=-51.442, rz=48.787, shoulder=lefty, elbow=epositive, wrist=wpositive, fatherId=fUserFrame[0]}
  [260] = {x=31.353, y=35.61, z=114.221, rx=180, ry=-52.756, rz=51.797, shoulder=lefty, elbow=epositive, wrist=wpositive, fatherId=fUserFrame[0]}
  [261] = {x=35.033, y=38.861, z=111.903, rx=180, ry=-54.096, rz=54.751, shoulder=lefty, elbow=epositive, wrist=wpositive, fatherId=fUserFrame[0]}
  [262] = {x=38.719, y=41.93, z=109.366, rx=180, ry=-55.456, rz=57.635, shoulder=lefty, elbow=epositive, wrist=wpositive, fatherId=fUserFrame[0]}
  [263] = {x=42.278, y=44.785, z=106.677, rx=180, ry=-56.784, rz=60.421, shoulder=lefty, elbow=epositive, wrist=wpositive, fatherId=fUserFrame[0]}
  [264] = {x=45.697, y=47.475, z=103.838, rx=180, ry=-58.069, rz=63.15, shoulder=lefty, elbow=epositive, wrist=wpositive, fatherId=fUserFrame[0]}
  [265] = {x=49.013, y=50.027, z=100.834, rx=180, ry=-59.331, rz=65.846, shoulder=lefty, elbow=epositive, wrist=wpositive, fatherId=fUserFrame[0]}
  [266] = {x=44.083, y=48.91, z=103.812, rx=180, ry=-56.777, rz=64.614, shoulder=lefty, elbow=epositive, wrist=wpositive, fatherId=fUserFrame[0]}
  [267] = {x=38.578, y=47.741, z=106.69, rx=180, ry=-54.005, rz=63.35, shoulder=lefty, elbow=epositive, wrist=wpositive, fatherId=fUserFrame[0]}
  [268] = {x=33.15, y=46.43, z=109.226, rx=180, ry=-51.395, rz=61.971, shoulder=lefty, elbow=epositive, wrist=wpositive, fatherId=fUserFrame[0]}
  [269] = {x=27.673, y=45.016, z=111.467, rx=180, ry=-48.846, rz=60.521, shoulder=lefty, elbow=epositive, wrist=wpositive, fatherId=fUserFrame[0]}
  [270] = {x=22.349, y=43.394, z=113.421, rx=180, ry=-46.48, rz=58.908, shoulder=lefty, elbow=epositive, wrist=wpositive, fatherId=fUserFrame[0]}
  [271] = {x=16.731, y=41.59, z=115.171, rx=180, ry=-44.042, rz=57.164, shoulder=lefty, elbow=epositive, wrist=wpositive, fatherId=fUserFrame[0]}
  [272] = {x=10.985, y=39.551, z=116.679, rx=180, ry=-41.623, rz=55.249, shoulder=lefty, elbow=epositive, wrist=wpositive, fatherId=fUserFrame[0]}
  [273] = {x=5.01, y=37.376, z=117.894, rx=180, ry=-39.136, rz=53.253, shoulder=lefty, elbow=epositive, wrist=wpositive, fatherId=fUserFrame[0]}
  [274] = {x=-0.804, y=35.019, z=118.802, rx=180, ry=-36.769, rz=51.14, shoulder=lefty, elbow=epositive, wrist=wpositive, fatherId=fUserFrame[0]}
  [275] = {x=-6.341, y=32.513, z=119.42, rx=180, ry=-34.555, rz=48.942, shoulder=lefty, elbow=epositive, wrist=wpositive, fatherId=fUserFrame[0]}
  [276] = {x=-11.541, y=29.826, z=119.795, rx=180, ry=-32.512, rz=46.633, shoulder=lefty, elbow=epositive, wrist=wpositive, fatherId=fUserFrame[0]}
  [277] = {x=-16.328, y=26.961, z=119.972, rx=180, ry=-30.663, rz=44.22, shoulder=lefty, elbow=epositive, wrist=wpositive, fatherId=fUserFrame[0]}
  [278] = {x=-20.759, y=23.89, z=119.984, rx=180, ry=-28.97, rz=41.681, shoulder=lefty, elbow=epositive, wrist=wpositive, fatherId=fUserFrame[0]}
  [279] = {x=-24.662, y=20.615, z=119.891, rx=180, ry=-27.501, rz=39.02, shoulder=lefty, elbow=epositive, wrist=wpositive, fatherId=fUserFrame[0]}
  [280] = {x=-28.137, y=17.281, z=119.682, rx=180, ry=-26.181, rz=36.344, shoulder=lefty, elbow=epositive, wrist=wpositive, fatherId=fUserFrame[0]}
  [281] = {x=-30.954, y=14.026, z=119.435, rx=180, ry=-25.107, rz=33.749, shoulder=lefty, elbow=epositive, wrist=wpositive, fatherId=fUserFrame[0]}
  [282] = {x=-33.378, y=10.884, z=119.125, rx=180, ry=-24.152, rz=31.253, shoulder=lefty, elbow=epositive, wrist=wpositive, fatherId=fUserFrame[0]}
  [283] = {x=-35.18, y=7.837, z=118.856, rx=180, ry=-23.436, rz=28.836, shoulder=lefty, elbow=epositive, wrist=wpositive, fatherId=fUserFrame[0]}
  [284] = {x=-36.701, y=4.771, z=118.561, rx=180, ry=-22.799, rz=26.415, shoulder=lefty, elbow=epositive, wrist=wpositive, fatherId=fUserFrame[0]}
  [285] = {x=-37.634, y=1.68, z=118.351, rx=180, ry=-22.393, rz=23.979, shoulder=lefty, elbow=epositive, wrist=wpositive, fatherId=fUserFrame[0]}
  [286] = {x=-31.685, y=1.329, z=120.133, rx=180, ry=-25.334, rz=23.724, shoulder=lefty, elbow=epositive, wrist=wpositive, fatherId=fUserFrame[0]}
  [287] = {x=-28.486, y=1.091, z=120.955, rx=180, ry=-26.896, rz=23.548, shoulder=lefty, elbow=epositive, wrist=wpositive, fatherId=fUserFrame[0]}
  [288] = {x=-25.13, y=0.851, z=121.716, rx=180, ry=-28.521, rz=23.371, shoulder=lefty, elbow=epositive, wrist=wpositive, fatherId=fUserFrame[0]}
  [289] = {x=-21.648, y=0.56, z=122.401, rx=180, ry=-30.194, rz=23.155, shoulder=lefty, elbow=epositive, wrist=wpositive, fatherId=fUserFrame[0]}
  [290] = {x=-17.999, y=0.268, z=123.005, rx=180, ry=-31.937, rz=22.938, shoulder=lefty, elbow=epositive, wrist=wpositive, fatherId=fUserFrame[0]}
  [291] = {x=-14.2, y=-0.07, z=123.512, rx=180, ry=-33.74, rz=22.686, shoulder=lefty, elbow=epositive, wrist=wpositive, fatherId=fUserFrame[0]}
  [292] = {x=-10.214, y=-0.41, z=123.912, rx=180, ry=-35.624, rz=22.432, shoulder=lefty, elbow=epositive, wrist=wpositive, fatherId=fUserFrame[0]}
  [293] = {x=-6.064, y=-0.79, z=124.188, rx=180, ry=-37.576, rz=22.148, shoulder=lefty, elbow=epositive, wrist=wpositive, fatherId=fUserFrame[0]}
  [294] = {x=-1.901, y=-1.162, z=124.321, rx=180, ry=-39.531, rz=21.87, shoulder=lefty, elbow=epositive, wrist=wpositive, fatherId=fUserFrame[0]}
  [295] = {x=2.184, y=-1.553, z=124.312, rx=180, ry=-41.448, rz=21.577, shoulder=lefty, elbow=epositive, wrist=wpositive, fatherId=fUserFrame[0]}
  [296] = {x=6.214, y=-1.935, z=124.167, rx=180, ry=-43.341, rz=21.29, shoulder=lefty, elbow=epositive, wrist=wpositive, fatherId=fUserFrame[0]}
  [297] = {x=10.181, y=-2.334, z=123.892, rx=180, ry=-45.206, rz=20.99, shoulder=lefty, elbow=epositive, wrist=wpositive, fatherId=fUserFrame[0]}
  [298] = {x=14.101, y=-2.726, z=123.491, rx=180, ry=-47.055, rz=20.695, shoulder=lefty, elbow=epositive, wrist=wpositive, fatherId=fUserFrame[0]}
  [299] = {x=17.978, y=-3.133, z=122.966, rx=180, ry=-48.89, rz=20.388, shoulder=lefty, elbow=epositive, wrist=wpositive, fatherId=fUserFrame[0]}
  [300] = {x=21.827, y=-3.535, z=122.317, rx=180, ry=-50.72, rz=20.086, shoulder=lefty, elbow=epositive, wrist=wpositive, fatherId=fUserFrame[0]}
  [301] = {x=25.648, y=-3.944, z=121.544, rx=180, ry=-52.547, rz=19.777, shoulder=lefty, elbow=epositive, wrist=wpositive, fatherId=fUserFrame[0]}
  [302] = {x=29.434, y=-4.346, z=120.65, rx=180, ry=-54.37, rz=19.474, shoulder=lefty, elbow=epositive, wrist=wpositive, fatherId=fUserFrame[0]}
  [303] = {x=33.191, y=-4.75, z=119.634, rx=180, ry=-56.193, rz=19.169, shoulder=lefty, elbow=epositive, wrist=wpositive, fatherId=fUserFrame[0]}
  [304] = {x=36.907, y=-5.147, z=118.499, rx=180, ry=-58.013, rz=18.869, shoulder=lefty, elbow=epositive, wrist=wpositive, fatherId=fUserFrame[0]}
  [305] = {x=36.9, y=-1.421, z=118.608, rx=180, ry=-58.063, rz=21.787, shoulder=lefty, elbow=epositive, wrist=wpositive, fatherId=fUserFrame[0]}
  [306] = {x=36.824, y=2.407, z=118.608, rx=180, ry=-58.029, rz=24.773, shoulder=lefty, elbow=epositive, wrist=wpositive, fatherId=fUserFrame[0]}
  [307] = {x=36.718, y=6.276, z=118.48, rx=180, ry=-57.927, rz=27.792, shoulder=lefty, elbow=epositive, wrist=wpositive, fatherId=fUserFrame[0]}
  [308] = {x=36.616, y=10.149, z=118.211, rx=180, ry=-57.771, rz=30.827, shoulder=lefty, elbow=epositive, wrist=wpositive, fatherId=fUserFrame[0]}
  [309] = {x=36.51, y=14.016, z=117.804, rx=180, ry=-57.557, rz=33.878, shoulder=lefty, elbow=epositive, wrist=wpositive, fatherId=fUserFrame[0]}
  [310] = {x=37.169, y=16.535, z=117.228, rx=180, ry=-57.751, rz=35.884, shoulder=lefty, elbow=epositive, wrist=wpositive, fatherId=fUserFrame[0]}
  [311] = {x=38.02, y=19.029, z=116.525, rx=180, ry=-58.02, rz=37.885, shoulder=lefty, elbow=epositive, wrist=wpositive, fatherId=fUserFrame[0]}
  [312] = {x=38.787, y=21.476, z=115.79, rx=180, ry=-58.228, rz=39.867, shoulder=lefty, elbow=epositive, wrist=wpositive, fatherId=fUserFrame[0]}
  [313] = {x=39.708, y=23.854, z=114.947, rx=180, ry=-58.501, rz=41.816, shoulder=lefty, elbow=epositive, wrist=wpositive, fatherId=fUserFrame[0]}
  [314] = {x=40.535, y=26.179, z=114.082, rx=180, ry=-58.709, rz=43.746, shoulder=lefty, elbow=epositive, wrist=wpositive, fatherId=fUserFrame[0]}
  [315] = {x=41.497, y=28.44, z=113.115, rx=180, ry=-58.976, rz=45.649, shoulder=lefty, elbow=epositive, wrist=wpositive, fatherId=fUserFrame[0]}
  [316] = {x=42.362, y=30.659, z=112.13, rx=180, ry=-59.176, rz=47.543, shoulder=lefty, elbow=epositive, wrist=wpositive, fatherId=fUserFrame[0]}
  [317] = {x=43.343, y=32.818, z=111.05, rx=180, ry=-59.428, rz=49.416, shoulder=lefty, elbow=epositive, wrist=wpositive, fatherId=fUserFrame[0]}
  [318] = {x=44.221, y=34.939, z=109.958, rx=180, ry=-59.61, rz=51.285, shoulder=lefty, elbow=epositive, wrist=wpositive, fatherId=fUserFrame[0]}
  [319] = {x=45.196, y=37.004, z=108.778, rx=180, ry=-59.834, rz=53.139, shoulder=lefty, elbow=epositive, wrist=wpositive, fatherId=fUserFrame[0]}
  [320] = {x=46.064, y=39.037, z=107.59, rx=180, ry=-59.985, rz=54.998, shoulder=lefty, elbow=epositive, wrist=wpositive, fatherId=fUserFrame[0]}
  [321] = {x=47.013, y=41.002, z=106.326, rx=180, ry=-60.173, rz=56.834, shoulder=lefty, elbow=epositive, wrist=wpositive, fatherId=fUserFrame[0]}
  [322] = {x=47.863, y=42.921, z=105.062, rx=180, ry=-60.293, rz=58.666, shoulder=lefty, elbow=epositive, wrist=wpositive, fatherId=fUserFrame[0]}
  [323] = {x=48.809, y=44.772, z=103.716, rx=180, ry=-60.46, rz=60.476, shoulder=lefty, elbow=epositive, wrist=wpositive, fatherId=fUserFrame[0]}
  [324] = {x=49.686, y=46.591, z=102.355, rx=180, ry=-60.572, rz=62.298, shoulder=lefty, elbow=epositive, wrist=wpositive, fatherId=fUserFrame[0]}
  [325] = {x=50.7, y=48.352, z=100.888, rx=180, ry=-60.754, rz=64.109, shoulder=lefty, elbow=epositive, wrist=wpositive, fatherId=fUserFrame[0]}
  [326] = {x=51.727, y=50.068, z=99.369, rx=180, ry=-60.931, rz=65.923, shoulder=lefty, elbow=epositive, wrist=wpositive, fatherId=fUserFrame[0]}
  [327] = {x=52.948, y=51.706, z=97.716, rx=180, ry=-61.221, rz=67.71, shoulder=lefty, elbow=epositive, wrist=wpositive, fatherId=fUserFrame[0]}
  [328] = {x=54.179, y=53.292, z=96.009, rx=180, ry=-61.51, rz=69.495, shoulder=lefty, elbow=epositive, wrist=wpositive, fatherId=fUserFrame[0]}
  [329] = {x=55.616, y=54.796, z=94.148, rx=180, ry=-61.931, rz=71.25, shoulder=lefty, elbow=epositive, wrist=wpositive, fatherId=fUserFrame[0]}
  [330] = {x=52.563, y=54.509, z=96.159, rx=180, ry=-60.128, rz=70.88, shoulder=lefty, elbow=epositive, wrist=wpositive, fatherId=fUserFrame[0]}
  [331] = {x=47.423, y=53.901, z=99.331, rx=180, ry=-57.206, rz=70.111, shoulder=lefty, elbow=epositive, wrist=wpositive, fatherId=fUserFrame[0]}
  [332] = {x=44.683, y=53.582, z=100.858, rx=180, ry=-55.691, rz=69.715, shoulder=lefty, elbow=epositive, wrist=wpositive, fatherId=fUserFrame[0]}
  [333] = {x=41.917, y=53.209, z=102.324, rx=180, ry=-54.209, rz=69.262, shoulder=lefty, elbow=epositive, wrist=wpositive, fatherId=fUserFrame[0]}
  [334] = {x=38.974, y=52.828, z=103.762, rx=180, ry=-52.655, rz=68.803, shoulder=lefty, elbow=epositive, wrist=wpositive, fatherId=fUserFrame[0]}
  [335] = {x=36.005, y=52.436, z=105.108, rx=180, ry=-51.115, rz=68.335, shoulder=lefty, elbow=epositive, wrist=wpositive, fatherId=fUserFrame[0]}
  [336] = {x=33.04, y=52.03, z=106.355, rx=180, ry=-49.603, rz=67.857, shoulder=lefty, elbow=epositive, wrist=wpositive, fatherId=fUserFrame[0]}
  [337] = {x=27.328, y=51.09, z=108.557, rx=180, ry=-46.799, rz=66.777, shoulder=lefty, elbow=epositive, wrist=wpositive, fatherId=fUserFrame[0]}
  [338] = {x=21.384, y=50.082, z=110.477, rx=180, ry=-43.956, rz=65.645, shoulder=lefty, elbow=epositive, wrist=wpositive, fatherId=fUserFrame[0]}
  [339] = {x=18.339, y=49.516, z=111.339, rx=180, ry=-42.539, rz=65.023, shoulder=lefty, elbow=epositive, wrist=wpositive, fatherId=fUserFrame[0]}
  [340] = {x=15.169, y=48.922, z=112.135, rx=180, ry=-41.078, rz=64.379, shoulder=lefty, elbow=epositive, wrist=wpositive, fatherId=fUserFrame[0]}
  [341] = {x=11.868, y=48.297, z=112.858, rx=180, ry=-39.57, rz=63.711, shoulder=lefty, elbow=epositive, wrist=wpositive, fatherId=fUserFrame[0]}
  [342] = {x=8.507, y=47.631, z=113.495, rx=180, ry=-38.055, rz=63.011, shoulder=lefty, elbow=epositive, wrist=wpositive, fatherId=fUserFrame[0]}
  [343] = {x=5.171, y=46.89, z=114.053, rx=180, ry=-36.584, rz=62.245, shoulder=lefty, elbow=epositive, wrist=wpositive, fatherId=fUserFrame[0]}
  [344] = {x=1.817, y=46.093, z=114.527, rx=180, ry=-35.126, rz=61.435, shoulder=lefty, elbow=epositive, wrist=wpositive, fatherId=fUserFrame[0]}
  [345] = {x=-1.542, y=45.234, z=114.917, rx=180, ry=-33.688, rz=60.577, shoulder=lefty, elbow=epositive, wrist=wpositive, fatherId=fUserFrame[0]}
  [346] = {x=-4.897, y=44.308, z=115.225, rx=180, ry=-32.273, rz=59.667, shoulder=lefty, elbow=epositive, wrist=wpositive, fatherId=fUserFrame[0]}
  [347] = {x=-11.566, y=42.2, z=115.614, rx=180, ry=-29.532, rz=57.648, shoulder=lefty, elbow=epositive, wrist=wpositive, fatherId=fUserFrame[0]}
  [348] = {x=-17.965, y=39.906, z=115.675, rx=180, ry=-26.955, rz=55.509, shoulder=lefty, elbow=epositive, wrist=wpositive, fatherId=fUserFrame[0]}
  [349] = {x=-24.031, y=37.42, z=115.459, rx=180, ry=-24.556, rz=53.247, shoulder=lefty, elbow=epositive, wrist=wpositive, fatherId=fUserFrame[0]}
  [350] = {x=-29.593, y=34.771, z=115.041, rx=180, ry=-22.399, rz=50.893, shoulder=lefty, elbow=epositive, wrist=wpositive, fatherId=fUserFrame[0]}
  [351] = {x=-34.725, y=31.939, z=114.463, rx=180, ry=-20.436, rz=48.431, shoulder=lefty, elbow=epositive, wrist=wpositive, fatherId=fUserFrame[0]}
  [352] = {x=-39.297, y=28.891, z=113.822, rx=180, ry=-18.731, rz=45.84, shoulder=lefty, elbow=epositive, wrist=wpositive, fatherId=fUserFrame[0]}
  [353] = {x=-43.448, y=25.6, z=113.12, rx=180, ry=-17.202, rz=43.1, shoulder=lefty, elbow=epositive, wrist=wpositive, fatherId=fUserFrame[0]}
  [354] = {x=-47.036, y=22.037, z=112.449, rx=180, ry=-15.915, rz=40.192, shoulder=lefty, elbow=epositive, wrist=wpositive, fatherId=fUserFrame[0]}
  [355] = {x=-50.183, y=18.336, z=111.758, rx=180, ry=-14.774, rz=37.218, shoulder=lefty, elbow=epositive, wrist=wpositive, fatherId=fUserFrame[0]}
  [356] = {x=-52.715, y=14.806, z=111.116, rx=180, ry=-13.835, rz=34.399, shoulder=lefty, elbow=epositive, wrist=wpositive, fatherId=fUserFrame[0]}
  [357] = {x=-52.715, y=14.806, z=161.116, rx=180, ry=-13.835, rz=34.399, shoulder=lefty, elbow=epositive, wrist=wpositive, fatherId=fUserFrame[0]}
  [358] = {x=4.278, y=3.411, z=174.216, rx=180, ry=-42.407, rz=-20.128, shoulder=lefty, elbow=epositive, wrist=wpositive, fatherId=fUserFrame[0]}
  [359] = {x=4.278, y=3.411, z=124.216, rx=180, ry=-42.407, rz=-20.128, shoulder=lefty, elbow=epositive, wrist=wpositive, fatherId=fUserFrame[0]}
  [360] = {x=3.791, y=-1.027, z=124.278, rx=180, ry=-42.212, rz=-23.599, shoulder=lefty, elbow=epositive, wrist=wpositive, fatherId=fUserFrame[0]}
  [361] = {x=4.289, y=-5.504, z=124.132, rx=180, ry=-42.386, rz=-27.1, shoulder=lefty, elbow=epositive, wrist=wpositive, fatherId=fUserFrame[0]}
  [362] = {x=5.782, y=-9.947, z=123.764, rx=180, ry=-42.934, rz=-30.59, shoulder=lefty, elbow=epositive, wrist=wpositive, fatherId=fUserFrame[0]}
  [363] = {x=8.224, y=-14.41, z=123.139, rx=180, ry=-43.84, rz=-34.117, shoulder=lefty, elbow=epositive, wrist=wpositive, fatherId=fUserFrame[0]}
  [364] = {x=11.501, y=-18.894, z=122.2, rx=180, ry=-45.057, rz=-37.697, shoulder=lefty, elbow=epositive, wrist=wpositive, fatherId=fUserFrame[0]}
  [365] = {x=9.824, y=-14.861, z=122.959, rx=180, ry=-44.571, rz=-34.478, shoulder=lefty, elbow=epositive, wrist=wpositive, fatherId=fUserFrame[0]}
  [366] = {x=8.613, y=-10.87, z=123.51, rx=180, ry=-44.23, rz=-31.322, shoulder=lefty, elbow=epositive, wrist=wpositive, fatherId=fUserFrame[0]}
  [367] = {x=7.921, y=-6.919, z=123.87, rx=180, ry=-44.06, rz=-28.217, shoulder=lefty, elbow=epositive, wrist=wpositive, fatherId=fUserFrame[0]}
  [368] = {x=7.772, y=-2.954, z=124.054, rx=180, ry=-44.073, rz=-25.116, shoulder=lefty, elbow=epositive, wrist=wpositive, fatherId=fUserFrame[0]}
  [369] = {x=8.16, y=0.997, z=124.064, rx=180, ry=-44.266, rz=-22.03, shoulder=lefty, elbow=epositive, wrist=wpositive, fatherId=fUserFrame[0]}
  [370] = {x=7.987, y=-2.551, z=124.05, rx=180, ry=-44.179, rz=-24.802, shoulder=lefty, elbow=epositive, wrist=wpositive, fatherId=fUserFrame[0]}
  [371] = {x=8.556, y=-6.099, z=123.875, rx=180, ry=-44.383, rz=-27.577, shoulder=lefty, elbow=epositive, wrist=wpositive, fatherId=fUserFrame[0]}
  [372] = {x=9.86, y=-9.613, z=123.529, rx=180, ry=-44.879, rz=-30.336, shoulder=lefty, elbow=epositive, wrist=wpositive, fatherId=fUserFrame[0]}
  [373] = {x=11.866, y=-13.123, z=122.992, rx=180, ry=-45.653, rz=-33.107, shoulder=lefty, elbow=epositive, wrist=wpositive, fatherId=fUserFrame[0]}
  [374] = {x=14.502, y=-16.628, z=122.234, rx=180, ry=-46.679, rz=-35.893, shoulder=lefty, elbow=epositive, wrist=wpositive, fatherId=fUserFrame[0]}
  [375] = {x=17.496, y=-20.822, z=121.12, rx=180, ry=-47.769, rz=-39.263, shoulder=lefty, elbow=epositive, wrist=wpositive, fatherId=fUserFrame[0]}
  [376] = {x=20.739, y=-24.824, z=119.755, rx=180, ry=-48.936, rz=-42.54, shoulder=lefty, elbow=epositive, wrist=wpositive, fatherId=fUserFrame[0]}
  [377] = {x=24.162, y=-28.607, z=118.15, rx=180, ry=-50.165, rz=-45.707, shoulder=lefty, elbow=epositive, wrist=wpositive, fatherId=fUserFrame[0]}
  [378] = {x=27.716, y=-32.196, z=116.305, rx=180, ry=-51.442, rz=-48.787, shoulder=lefty, elbow=epositive, wrist=wpositive, fatherId=fUserFrame[0]}
  [379] = {x=31.353, y=-35.61, z=114.221, rx=180, ry=-52.756, rz=-51.797, shoulder=lefty, elbow=epositive, wrist=wpositive, fatherId=fUserFrame[0]}
  [380] = {x=35.033, y=-38.861, z=111.903, rx=180, ry=-54.096, rz=-54.751, shoulder=lefty, elbow=epositive, wrist=wpositive, fatherId=fUserFrame[0]}
  [381] = {x=38.719, y=-41.93, z=109.366, rx=180, ry=-55.456, rz=-57.635, shoulder=lefty, elbow=epositive, wrist=wpositive, fatherId=fUserFrame[0]}
  [382] = {x=42.278, y=-44.785, z=106.677, rx=180, ry=-56.784, rz=-60.421, shoulder=lefty, elbow=epositive, wrist=wpositive, fatherId=fUserFrame[0]}
  [383] = {x=45.697, y=-47.475, z=103.838, rx=180, ry=-58.069, rz=-63.15, shoulder=lefty, elbow=epositive, wrist=wpositive, fatherId=fUserFrame[0]}
  [384] = {x=49.013, y=-50.027, z=100.834, rx=180, ry=-59.331, rz=-65.846, shoulder=lefty, elbow=epositive, wrist=wpositive, fatherId=fUserFrame[0]}
  [385] = {x=44.083, y=-48.91, z=103.812, rx=180, ry=-56.777, rz=-64.614, shoulder=lefty, elbow=epositive, wrist=wpositive, fatherId=fUserFrame[0]}
  [386] = {x=38.578, y=-47.741, z=106.69, rx=180, ry=-54.005, rz=-63.35, shoulder=lefty, elbow=epositive, wrist=wpositive, fatherId=fUserFrame[0]}
  [387] = {x=33.15, y=-46.43, z=109.226, rx=180, ry=-51.395, rz=-61.971, shoulder=lefty, elbow=epositive, wrist=wpositive, fatherId=fUserFrame[0]}
  [388] = {x=27.673, y=-45.016, z=111.467, rx=180, ry=-48.846, rz=-60.521, shoulder=lefty, elbow=epositive, wrist=wpositive, fatherId=fUserFrame[0]}
  [389] = {x=22.349, y=-43.394, z=113.421, rx=180, ry=-46.48, rz=-58.908, shoulder=lefty, elbow=epositive, wrist=wpositive, fatherId=fUserFrame[0]}
  [390] = {x=16.731, y=-41.59, z=115.171, rx=180, ry=-44.042, rz=-57.164, shoulder=lefty, elbow=epositive, wrist=wpositive, fatherId=fUserFrame[0]}
  [391] = {x=10.985, y=-39.551, z=116.679, rx=180, ry=-41.623, rz=-55.249, shoulder=lefty, elbow=epositive, wrist=wpositive, fatherId=fUserFrame[0]}
  [392] = {x=5.01, y=-37.376, z=117.894, rx=180, ry=-39.136, rz=-53.253, shoulder=lefty, elbow=epositive, wrist=wpositive, fatherId=fUserFrame[0]}
  [393] = {x=-0.804, y=-35.019, z=118.802, rx=180, ry=-36.769, rz=-51.14, shoulder=lefty, elbow=epositive, wrist=wpositive, fatherId=fUserFrame[0]}
  [394] = {x=-6.341, y=-32.513, z=119.42, rx=180, ry=-34.555, rz=-48.942, shoulder=lefty, elbow=epositive, wrist=wpositive, fatherId=fUserFrame[0]}
  [395] = {x=-11.541, y=-29.826, z=119.795, rx=180, ry=-32.512, rz=-46.633, shoulder=lefty, elbow=epositive, wrist=wpositive, fatherId=fUserFrame[0]}
  [396] = {x=-16.328, y=-26.961, z=119.972, rx=180, ry=-30.663, rz=-44.22, shoulder=lefty, elbow=epositive, wrist=wpositive, fatherId=fUserFrame[0]}
  [397] = {x=-20.759, y=-23.89, z=119.984, rx=180, ry=-28.97, rz=-41.681, shoulder=lefty, elbow=epositive, wrist=wpositive, fatherId=fUserFrame[0]}
  [398] = {x=-24.662, y=-20.615, z=119.891, rx=180, ry=-27.501, rz=-39.02, shoulder=lefty, elbow=epositive, wrist=wpositive, fatherId=fUserFrame[0]}
  [399] = {x=-28.137, y=-17.281, z=119.682, rx=180, ry=-26.181, rz=-36.344, shoulder=lefty, elbow=epositive, wrist=wpositive, fatherId=fUserFrame[0]}
  [400] = {x=-30.954, y=-14.026, z=119.435, rx=180, ry=-25.107, rz=-33.749, shoulder=lefty, elbow=epositive, wrist=wpositive, fatherId=fUserFrame[0]}
  [401] = {x=-33.378, y=-10.884, z=119.125, rx=180, ry=-24.152, rz=-31.253, shoulder=lefty, elbow=epositive, wrist=wpositive, fatherId=fUserFrame[0]}
  [402] = {x=-35.18, y=-7.837, z=118.856, rx=180, ry=-23.436, rz=-28.836, shoulder=lefty, elbow=epositive, wrist=wpositive, fatherId=fUserFrame[0]}
  [403] = {x=-36.701, y=-4.771, z=118.561, rx=180, ry=-22.799, rz=-26.415, shoulder=lefty, elbow=epositive, wrist=wpositive, fatherId=fUserFrame[0]}
  [404] = {x=-37.634, y=-1.68, z=118.351, rx=180, ry=-22.393, rz=-23.979, shoulder=lefty, elbow=epositive, wrist=wpositive, fatherId=fUserFrame[0]}
  [405] = {x=-31.685, y=-1.329, z=120.133, rx=180, ry=-25.334, rz=-23.724, shoulder=lefty, elbow=epositive, wrist=wpositive, fatherId=fUserFrame[0]}
  [406] = {x=-28.486, y=-1.091, z=120.955, rx=180, ry=-26.896, rz=-23.548, shoulder=lefty, elbow=epositive, wrist=wpositive, fatherId=fUserFrame[0]}
  [407] = {x=-25.13, y=-0.851, z=121.716, rx=180, ry=-28.521, rz=-23.371, shoulder=lefty, elbow=epositive, wrist=wpositive, fatherId=fUserFrame[0]}
  [408] = {x=-21.648, y=-0.56, z=122.401, rx=180, ry=-30.194, rz=-23.155, shoulder=lefty, elbow=epositive, wrist=wpositive, fatherId=fUserFrame[0]}
  [409] = {x=-17.999, y=-0.268, z=123.005, rx=180, ry=-31.937, rz=-22.938, shoulder=lefty, elbow=epositive, wrist=wpositive, fatherId=fUserFrame[0]}
  [410] = {x=-14.2, y=0.07, z=123.512, rx=180, ry=-33.74, rz=-22.686, shoulder=lefty, elbow=epositive, wrist=wpositive, fatherId=fUserFrame[0]}
  [411] = {x=-10.214, y=0.41, z=123.912, rx=180, ry=-35.624, rz=-22.432, shoulder=lefty, elbow=epositive, wrist=wpositive, fatherId=fUserFrame[0]}
  [412] = {x=-6.064, y=0.79, z=124.188, rx=180, ry=-37.576, rz=-22.148, shoulder=lefty, elbow=epositive, wrist=wpositive, fatherId=fUserFrame[0]}
  [413] = {x=-1.901, y=1.162, z=124.321, rx=180, ry=-39.531, rz=-21.87, shoulder=lefty, elbow=epositive, wrist=wpositive, fatherId=fUserFrame[0]}
  [414] = {x=2.184, y=1.553, z=124.312, rx=180, ry=-41.448, rz=-21.577, shoulder=lefty, elbow=epositive, wrist=wpositive, fatherId=fUserFrame[0]}
  [415] = {x=6.214, y=1.935, z=124.167, rx=180, ry=-43.341, rz=-21.29, shoulder=lefty, elbow=epositive, wrist=wpositive, fatherId=fUserFrame[0]}
  [416] = {x=10.181, y=2.334, z=123.892, rx=180, ry=-45.206, rz=-20.99, shoulder=lefty, elbow=epositive, wrist=wpositive, fatherId=fUserFrame[0]}
  [417] = {x=14.101, y=2.726, z=123.491, rx=180, ry=-47.055, rz=-20.695, shoulder=lefty, elbow=epositive, wrist=wpositive, fatherId=fUserFrame[0]}
  [418] = {x=17.978, y=3.133, z=122.966, rx=180, ry=-48.89, rz=-20.388, shoulder=lefty, elbow=epositive, wrist=wpositive, fatherId=fUserFrame[0]}
  [419] = {x=21.827, y=3.535, z=122.317, rx=180, ry=-50.72, rz=-20.086, shoulder=lefty, elbow=epositive, wrist=wpositive, fatherId=fUserFrame[0]}
  [420] = {x=25.648, y=3.944, z=121.544, rx=180, ry=-52.547, rz=-19.777, shoulder=lefty, elbow=epositive, wrist=wpositive, fatherId=fUserFrame[0]}
  [421] = {x=29.434, y=4.346, z=120.65, rx=180, ry=-54.37, rz=-19.474, shoulder=lefty, elbow=epositive, wrist=wpositive, fatherId=fUserFrame[0]}
  [422] = {x=33.191, y=4.75, z=119.634, rx=180, ry=-56.193, rz=-19.169, shoulder=lefty, elbow=epositive, wrist=wpositive, fatherId=fUserFrame[0]}
  [423] = {x=36.907, y=5.147, z=118.499, rx=180, ry=-58.013, rz=-18.869, shoulder=lefty, elbow=epositive, wrist=wpositive, fatherId=fUserFrame[0]}
  [424] = {x=36.9, y=1.421, z=118.608, rx=180, ry=-58.063, rz=-21.787, shoulder=lefty, elbow=epositive, wrist=wpositive, fatherId=fUserFrame[0]}
  [425] = {x=36.824, y=-2.407, z=118.608, rx=180, ry=-58.029, rz=-24.773, shoulder=lefty, elbow=epositive, wrist=wpositive, fatherId=fUserFrame[0]}
  [426] = {x=36.718, y=-6.276, z=118.48, rx=180, ry=-57.927, rz=-27.792, shoulder=lefty, elbow=epositive, wrist=wpositive, fatherId=fUserFrame[0]}
  [427] = {x=36.616, y=-10.149, z=118.211, rx=180, ry=-57.771, rz=-30.827, shoulder=lefty, elbow=epositive, wrist=wpositive, fatherId=fUserFrame[0]}
  [428] = {x=36.51, y=-14.016, z=117.804, rx=180, ry=-57.557, rz=-33.878, shoulder=lefty, elbow=epositive, wrist=wpositive, fatherId=fUserFrame[0]}
  [429] = {x=37.169, y=-16.535, z=117.228, rx=180, ry=-57.751, rz=-35.884, shoulder=lefty, elbow=epositive, wrist=wpositive, fatherId=fUserFrame[0]}
  [430] = {x=38.02, y=-19.029, z=116.525, rx=180, ry=-58.02, rz=-37.885, shoulder=lefty, elbow=epositive, wrist=wpositive, fatherId=fUserFrame[0]}
  [431] = {x=38.787, y=-21.476, z=115.79, rx=180, ry=-58.228, rz=-39.867, shoulder=lefty, elbow=epositive, wrist=wpositive, fatherId=fUserFrame[0]}
  [432] = {x=39.708, y=-23.854, z=114.947, rx=180, ry=-58.501, rz=-41.816, shoulder=lefty, elbow=epositive, wrist=wpositive, fatherId=fUserFrame[0]}
  [433] = {x=40.535, y=-26.179, z=114.082, rx=180, ry=-58.709, rz=-43.746, shoulder=lefty, elbow=epositive, wrist=wpositive, fatherId=fUserFrame[0]}
  [434] = {x=41.497, y=-28.44, z=113.115, rx=180, ry=-58.976, rz=-45.649, shoulder=lefty, elbow=epositive, wrist=wpositive, fatherId=fUserFrame[0]}
  [435] = {x=42.362, y=-30.659, z=112.13, rx=180, ry=-59.176, rz=-47.543, shoulder=lefty, elbow=epositive, wrist=wpositive, fatherId=fUserFrame[0]}
  [436] = {x=43.343, y=-32.818, z=111.05, rx=180, ry=-59.428, rz=-49.416, shoulder=lefty, elbow=epositive, wrist=wpositive, fatherId=fUserFrame[0]}
  [437] = {x=44.221, y=-34.939, z=109.958, rx=180, ry=-59.61, rz=-51.285, shoulder=lefty, elbow=epositive, wrist=wpositive, fatherId=fUserFrame[0]}
  [438] = {x=45.196, y=-37.004, z=108.778, rx=180, ry=-59.834, rz=-53.139, shoulder=lefty, elbow=epositive, wrist=wpositive, fatherId=fUserFrame[0]}
  [439] = {x=46.064, y=-39.037, z=107.59, rx=180, ry=-59.985, rz=-54.998, shoulder=lefty, elbow=epositive, wrist=wpositive, fatherId=fUserFrame[0]}
  [440] = {x=47.013, y=-41.002, z=106.326, rx=180, ry=-60.173, rz=-56.834, shoulder=lefty, elbow=epositive, wrist=wpositive, fatherId=fUserFrame[0]}
  [441] = {x=47.863, y=-42.921, z=105.062, rx=180, ry=-60.293, rz=-58.666, shoulder=lefty, elbow=epositive, wrist=wpositive, fatherId=fUserFrame[0]}
  [442] = {x=48.809, y=-44.772, z=103.716, rx=180, ry=-60.46, rz=-60.476, shoulder=lefty, elbow=epositive, wrist=wpositive, fatherId=fUserFrame[0]}
  [443] = {x=49.686, y=-46.591, z=102.355, rx=180, ry=-60.572, rz=-62.298, shoulder=lefty, elbow=epositive, wrist=wpositive, fatherId=fUserFrame[0]}
  [444] = {x=50.7, y=-48.352, z=100.888, rx=180, ry=-60.754, rz=-64.109, shoulder=lefty, elbow=epositive, wrist=wpositive, fatherId=fUserFrame[0]}
  [445] = {x=51.727, y=-50.068, z=99.369, rx=180, ry=-60.931, rz=-65.923, shoulder=lefty, elbow=epositive, wrist=wpositive, fatherId=fUserFrame[0]}
  [446] = {x=52.948, y=-51.706, z=97.716, rx=180, ry=-61.221, rz=-67.71, shoulder=lefty, elbow=epositive, wrist=wpositive, fatherId=fUserFrame[0]}
  [447] = {x=54.179, y=-53.292, z=96.009, rx=180, ry=-61.51, rz=-69.495, shoulder=lefty, elbow=epositive, wrist=wpositive, fatherId=fUserFrame[0]}
  [448] = {x=55.616, y=-54.796, z=94.148, rx=180, ry=-61.931, rz=-71.25, shoulder=lefty, elbow=epositive, wrist=wpositive, fatherId=fUserFrame[0]}
  [449] = {x=52.563, y=-54.509, z=96.159, rx=180, ry=-60.128, rz=-70.88, shoulder=lefty, elbow=epositive, wrist=wpositive, fatherId=fUserFrame[0]}
  [450] = {x=47.423, y=-53.901, z=99.331, rx=180, ry=-57.206, rz=-70.111, shoulder=lefty, elbow=epositive, wrist=wpositive, fatherId=fUserFrame[0]}
  [451] = {x=44.683, y=-53.582, z=100.858, rx=180, ry=-55.691, rz=-69.715, shoulder=lefty, elbow=epositive, wrist=wpositive, fatherId=fUserFrame[0]}
  [452] = {x=41.917, y=-53.209, z=102.324, rx=180, ry=-54.209, rz=-69.262, shoulder=lefty, elbow=epositive, wrist=wpositive, fatherId=fUserFrame[0]}
  [453] = {x=38.974, y=-52.828, z=103.762, rx=180, ry=-52.655, rz=-68.803, shoulder=lefty, elbow=epositive, wrist=wpositive, fatherId=fUserFrame[0]}
  [454] = {x=36.005, y=-52.436, z=105.108, rx=180, ry=-51.115, rz=-68.335, shoulder=lefty, elbow=epositive, wrist=wpositive, fatherId=fUserFrame[0]}
  [455] = {x=33.04, y=-52.03, z=106.355, rx=180, ry=-49.603, rz=-67.857, shoulder=lefty, elbow=epositive, wrist=wpositive, fatherId=fUserFrame[0]}
  [456] = {x=27.328, y=-51.09, z=108.557, rx=180, ry=-46.799, rz=-66.777, shoulder=lefty, elbow=epositive, wrist=wpositive, fatherId=fUserFrame[0]}
  [457] = {x=21.384, y=-50.082, z=110.477, rx=180, ry=-43.956, rz=-65.645, shoulder=lefty, elbow=epositive, wrist=wpositive, fatherId=fUserFrame[0]}
  [458] = {x=18.339, y=-49.516, z=111.339, rx=180, ry=-42.539, rz=-65.023, shoulder=lefty, elbow=epositive, wrist=wpositive, fatherId=fUserFrame[0]}
  [459] = {x=15.169, y=-48.922, z=112.135, rx=180, ry=-41.078, rz=-64.379, shoulder=lefty, elbow=epositive, wrist=wpositive, fatherId=fUserFrame[0]}
  [460] = {x=11.868, y=-48.297, z=112.858, rx=180, ry=-39.57, rz=-63.711, shoulder=lefty, elbow=epositive, wrist=wpositive, fatherId=fUserFrame[0]}
  [461] = {x=8.507, y=-47.631, z=113.495, rx=180, ry=-38.055, rz=-63.011, shoulder=lefty, elbow=epositive, wrist=wpositive, fatherId=fUserFrame[0]}
  [462] = {x=5.171, y=-46.89, z=114.053, rx=180, ry=-36.584, rz=-62.245, shoulder=lefty, elbow=epositive, wrist=wpositive, fatherId=fUserFrame[0]}
  [463] = {x=1.817, y=-46.093, z=114.527, rx=180, ry=-35.126, rz=-61.435, shoulder=lefty, elbow=epositive, wrist=wpositive, fatherId=fUserFrame[0]}
  [464] = {x=-1.542, y=-45.234, z=114.917, rx=180, ry=-33.688, rz=-60.577, shoulder=lefty, elbow=epositive, wrist=wpositive, fatherId=fUserFrame[0]}
  [465] = {x=-4.897, y=-44.308, z=115.225, rx=180, ry=-32.273, rz=-59.667, shoulder=lefty, elbow=epositive, wrist=wpositive, fatherId=fUserFrame[0]}
  [466] = {x=-11.566, y=-42.2, z=115.614, rx=180, ry=-29.532, rz=-57.648, shoulder=lefty, elbow=epositive, wrist=wpositive, fatherId=fUserFrame[0]}
  [467] = {x=-17.965, y=-39.906, z=115.675, rx=180, ry=-26.955, rz=-55.509, shoulder=lefty, elbow=epositive, wrist=wpositive, fatherId=fUserFrame[0]}
  [468] = {x=-24.031, y=-37.42, z=115.459, rx=180, ry=-24.556, rz=-53.247, shoulder=lefty, elbow=epositive, wrist=wpositive, fatherId=fUserFrame[0]}
  [469] = {x=-29.593, y=-34.771, z=115.041, rx=180, ry=-22.399, rz=-50.893, shoulder=lefty, elbow=epositive, wrist=wpositive, fatherId=fUserFrame[0]}
  [470] = {x=-34.725, y=-31.939, z=114.463, rx=180, ry=-20.436, rz=-48.431, shoulder=lefty, elbow=epositive, wrist=wpositive, fatherId=fUserFrame[0]}
  [471] = {x=-39.297, y=-28.891, z=113.822, rx=180, ry=-18.731, rz=-45.84, shoulder=lefty, elbow=epositive, wrist=wpositive, fatherId=fUserFrame[0]}
  [472] = {x=-43.448, y=-25.6, z=113.12, rx=180, ry=-17.202, rz=-43.1, shoulder=lefty, elbow=epositive, wrist=wpositive, fatherId=fUserFrame[0]}
  [473] = {x=-47.036, y=-22.037, z=112.449, rx=180, ry=-15.915, rz=-40.192, shoulder=lefty, elbow=epositive, wrist=wpositive, fatherId=fUserFrame[0]}
  [474] = {x=-50.183, y=-18.336, z=111.758, rx=180, ry=-14.774, rz=-37.218, shoulder=lefty, elbow=epositive, wrist=wpositive, fatherId=fUserFrame[0]}
  [475] = {x=-52.715, y=-14.806, z=111.116, rx=180, ry=-13.835, rz=-34.399, shoulder=lefty, elbow=epositive, wrist=wpositive, fatherId=fUserFrame[0]}
  [476] = {x=-52.715, y=-14.806, z=161.116, rx=180, ry=-13.835, rz=-34.399, shoulder=lefty, elbow=epositive, wrist=wpositive, fatherId=fUserFrame[0]}
  [477] = {x=-39.284, y=-14.806, z=215.651, rx=180, ry=-13.835, rz=-34.399, shoulder=lefty, elbow=epositive, wrist=wpositive, fatherId=fUserFrame[0]}
public tool tTool = {fatherId=flange[0], ioLink=valve1}
